// Mitsubishi GX Works2 project: 42015054   PLC: Q02/Q02H
// 42015054

PROGRAM MAIN
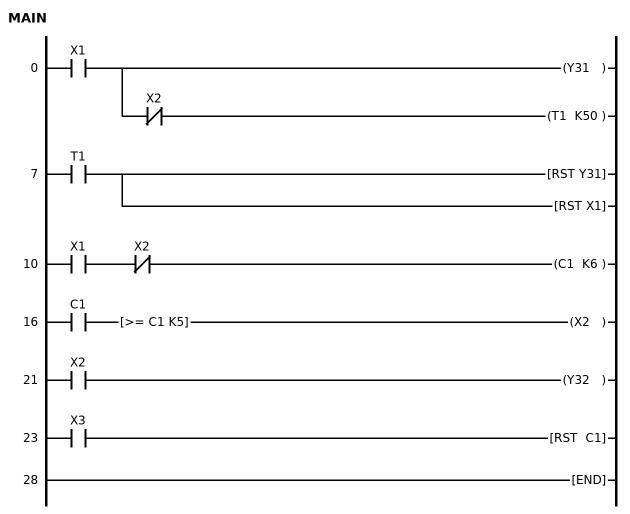
0     LD      X1
      OUT     Y31
      ANI     X2
      OUT     T1 K50
7     LD      T1
      RST     Y31
      RST     X1
10    LD      X1
      ANI     X2
      OUT     C1 K6
16    LD      C1
      AND>=   C1 K5
      OUT     X2
21    LD      X2
      OUT     Y32
23    LD      X3
      RST     C1
28    END
END_PROGRAM
